(* CODESYS project FB_Build_tcpdump_capture.export

Project tree, tasks and I/O mapping:
  function block FbBuildBashCommand [ST]
*)

// FbBuildBashCommand
FUNCTION_BLOCK FbBuildBashCommand
VAR_INPUT
	sProgramm: STRING(7) := 'tcpdump';
	sInterface: STRING(6) := '-i br0';
	// '/media/sd/' for SD card
	// '/var/www/' for flash and dwonload via WBM
	sFileLocation: STRING := '/media/sd/';
	sFileName: STRING := 'br0_capture';
	(*  Used ports by PFC 
		Port 22			-- Secure Shell SSH
		Port 23			-- Telnet
		Port 25			-- SMTP Mail routing
		Port 123		-- SNTP
		Port 80, 8080	--  HTTP
		Port 443		-- HTTPS
		Port 161,162	-- SNMP
		Port 44818		-- Ethernet/IP TCP Port
		Port 2222		-- Ethernet/IP UDP Port
		Port 502		-- Modbus TCP / UDP Port
		Port 2000		-- Modbus TCP / UDP Port WagoAppPLCModbus
		Port 6626		-- Wago Services
		Port 2455		-- Codesys 2.3
		Port 11740		-- Codesys 3 (e!Runtime)
		Port 67			-- DHCP / BootP Server Port
		Port 68			-- BootP / DHCP Port
		Port 1194		-- OpenVPN
		Port 1293		-- IPSec
		Port 1883		-- MQTT (Unencrypted)
		Port 8883		-- MQTT (Encrypted)
		Port 4840		-- OPC UA
	*)
	sCaputrePort: STRING := '11470';
END_VAR
VAR
	
	
	
END_VAR

VAR_OUTPUT
strCommand:STRING;

END_VAR

strCommand:=Format9(
	sFormat:= '%s %s %s %s%s%s %s %s &', 
	p1:=ADR(sProgramm) , 
	p2:=ADR(sInterface) , 
	p3:=ADR('-w') , 
	p4:=ADR(sFileLocation) , 
	p5:=ADR(sFileName) , 
	p6:=ADR('.pcap'), 
	p7:=ADR(' port'), 
	p8:=ADR(sCaputrePort) , 
	p9:=ADR('') );

END_FUNCTION_BLOCK
